FUNCTION_BLOCK FB_Elevator
VAR
	Up,
	Down,
	Slow,
	Brake :BOOL;
END_VAR

ACTION MoveDown:
Up:=FALSE;
Down:=TRUE;
Slow:=FALSE;
Brake:=FALSE;
END_ACTION

ACTION MoveUp:
Up:=TRUE;
Down:=FALSE;
Slow:=FALSE;
Brake:=FALSE;
END_ACTION

ACTION SlowDown:
Slow:=TRUE;
END_ACTION

ACTION Stop:
Up:=
Down:=
Slow:=FALSE;
Brake:=TRUE;
END_ACTION

END_FUNCTION_BLOCK

(* stored: Version 1.1.0.1, ProductVersion 3.1.4024.11
   POU FB_Elevator: Id {5904b407-8b88-4e68-9b86-33a97d4ede29}, SpecialFunc None
   Action MoveDown: Id {fbd0998e-dc21-4137-8767-13118fd4f0cc}
   Action MoveUp: Id {c2141de1-4ac1-467b-82dc-e7696b654923}
   Action SlowDown: Id {22c806b6-d209-4e38-aa92-07440957d394}
   Action Stop: Id {0cbeb641-d90e-4562-8ccf-eaab96289ac5} *)
